PROGRAM MAIN
VAR
	fbXAxis : Axis;
	fbYAxis : Axis;
	fbZ1Axis : Axis;
	fbZ2Axis : Axis;
	
	bHomeZ1Z2Axis : BOOL;
	bHomeXYAxis : BOOL;
	bHomingStarted : BOOL;
	bDecoupleXYAxis : BOOL;
	diStep : DINT;
	sTLMqttName: STRING(8) := 'PLC_CHAN';
	messageIndex: UINT;
	stMqttPayload: MqttFramework.ST_MqttPayload;
	sMessage : STRING;
	evalIndex : INT;
END_VAR

fbXAxis();
fbYAxis();

IF bDecoupleXYAxis
THEN

	IF fbXAxis
		.PrepareDecoupling(fbYAxis.axisRef,fbYAxis.fbMcReadStatus.Status)
		.StartDecoupling()
	THEN
		//Decoupling successful
		bDecoupleXYAxis := FALSE;
	END_IF
	
END_IF

IF bHomeXYAxis
THEN
	
	IF fbXAxis
		.PrepareCoupling(fbYAxis.axisRef,fbYAxis.fbMcReadStatus.Status, -1, 1)
		.StartCoupling()
		.StartHoming()
	THEN
		bHomeXYAxis := FALSE;
		bHomingStarted := FALSE;
	END_IF
	
END_IF


CASE diStep OF
	
	0:
	
		IF ADS.fbMqttClient.Subscribe(sTopic := sTLMqttName)
		THEN			
			diStep := 10;
		END_IF
	
	
	10:
	
		messageIndex := ADS.fbMqttClient.isNewMessage(sTLMqttName);
		IF messageIndex > 0
		THEN
			stMqttPayload := Ads.fbMqttClient.getNewMessage(messageIndex);
			diStep:=20;
		END_IF
		
	//Payloadauswertung	
	20:
	
		sMessage := '';
		FOR evalIndex := 1 TO 32 DO
			sMessage := CONCAT(sMessage , F_ToCHR(stMqttPayload.data[evalIndex]));
		END_FOR
		
		diStep:=30;
	
	30:
	
		IF sMessage = 'cmd_home'
		THEN
			bHomeXYAxis := TRUE;
			diStep := 10;
		END_IF
	
END_CASE

END_PROGRAM

(* stored: Version 1.1.0.1, ProductVersion 3.1.4024.2
   POU MAIN: Id {94fb3a52-0038-400d-b211-29ede54e5f58}, SpecialFunc None *)
